Staubli VAL3: LineSymArray.pgx

public program LineSymArray(trsf& x_trSource[], trsf& x_trLine[], trsf& x_trDest[], bool& x_bRes)
  local num l_nNum
begin

  //点的数组有关直线对称
  for l_nNum=0 to size(x_trSource)-1
    call LineSym(x_trSource[l_nNum],x_trLine,x_trDest[l_nNum],x_bRes)
    if !x_bRes
      return
    endIf
  endFor
end
